# EPICS substitutions: odmApp/Db/odm-sys0-od01.substitutions
file MO2i.template
{
pattern	{ PRIM, LOCA, UNIT, PORT,         SCAN      }
		{ ODM,  LI00, 100,    OXI_$(LOCA), "1 second" }
		{ ODM,  LI01, 100,    OXI_$(LOCA), "1 second" }
		{ ODM,  LI02, 100,    OXI_$(LOCA), "1 second" }
		{ ODM,  LI03, 100,    OXI_$(LOCA), "1 second" }
		{ ODM,  LI04, 100,    OXI_$(LOCA), "1 second" }
		{ ODM,  LI05, 100,    OXI_$(LOCA), "1 second" }
		{ ODM,  LI06, 100,    OXI_$(LOCA), "1 second" }
		{ ODM,  LI07, 100,    OXI_$(LOCA), "1 second" }
		{ ODM,  LI08, 100,    OXI_$(LOCA), "1 second" }
}

file odm-oxigraf-alias.template
{
pattern	{ LOCA }
		{ LI00 }
		{ LI01 }
		{ LI02 }
		{ LI03 }
		{ LI04 }
		{ LI05 }
		{ LI06 }
		{ LI07 }
		{ LI08 }
}

file asynRecord.db
{
pattern{ P               , R          , PORT, ADDR, IMAX, OMAX }
		{ SIOC:LI00:OD01:, ASYNDRIVER , OXI_LI00,  0,0, 0    }
}

file sioc-sys0-od01.db
{
  {NULL=NULL}
}
